(* IEC 61131-3 sources: ics_security/plc_ladder_logic/programs, 9 files *)

(* ---- led_ladder_logic_bomb.st ---- *)
PROGRAM part1c
  VAR
    Input0 AT %IX1.0 : BOOL;
    Output0 AT %QX1.0 : BOOL;
  END_VAR
  VAR
    TP0 : TP;
    Trigger0 : BOOL;
    Trigger1 : BOOL;
    CTU0 : CTU;
    TON0 : TON;
    SR0 : SR;
    R_TRIG1 : R_TRIG;
  END_VAR

  TP0(IN := Input0, PT := T#6s);
  Output0 := Input0 OR TP0.Q OR Trigger0 OR Trigger1;
  R_TRIG1(CLK := Input0);
  CTU0(CU := R_TRIG1.Q, PV := 6);
  Trigger0 := CTU0.Q;
  TON0(IN := Input0, PT := T#30s);
  SR0(S1 := TON0.Q);
  Trigger1 := SR0.Q1;
  Output0 := NOT(NOT(Input0) AND NOT(Trigger1) AND NOT(Trigger0));
END_PROGRAM

CONFIGURATION Config0

  RESOURCE Res0 ON PLC
    TASK task0(INTERVAL := T#20ms,PRIORITY := 0);
    PROGRAM instance0 WITH task0 : part1c;
  END_RESOURCE
END_CONFIGURATION

(* ---- led_loop.st ---- *)
PROGRAM part1b
  VAR
    Input0 AT %IX1.0 : BOOL;
    Output0 AT %QX1.0 : BOOL;
  END_VAR
  VAR
    TP0 : TP;
  END_VAR

  TP0(IN := Input0, PT := T#6s);
  Output0 := TP0.Q;
  Output0 := Input0;
  Output0 := NOT(NOT(Input0));
END_PROGRAM

CONFIGURATION Config0

  RESOURCE Res0 ON PLC
    TASK task0(INTERVAL := T#20ms,PRIORITY := 0);
    PROGRAM instance0 WITH task0 : part1b;
  END_RESOURCE
END_CONFIGURATION

(* ---- led_switch_activated.st ---- *)
PROGRAM part1a
  VAR
    Input0 AT %IX1.0 : BOOL;
    Input1 AT %IX1.1 : BOOL;
    Output0 AT %QX1.0 : BOOL;
    Output1 AT %QX1.1 : BOOL;
  END_VAR

  Output1 := Input0;
  Output0 := NOT(Input1);
END_PROGRAM

CONFIGURATION Config0

  RESOURCE Res0 ON PLC
    TASK task0(INTERVAL := T#20ms,PRIORITY := 0);
    PROGRAM instance0 WITH task0 : part1a;
  END_RESOURCE
END_CONFIGURATION

(* ---- robot_path.st ---- *)
PROGRAM part2
  VAR
    pos_x0 AT %IX0.0 : BOOL;
    pos_x1 AT %IX0.1 : BOOL;
    pos_x2 AT %IX0.2 : BOOL;
    pos_x3 AT %IX0.3 : BOOL;
  END_VAR
  VAR
    pos_x : UINT;
  END_VAR
  VAR
    pos_y0 AT %IX0.4 : BOOL;
    pos_y1 AT %IX0.5 : BOOL;
    pos_y2 AT %IX0.6 : BOOL;
    pos_y3 AT %IX0.7 : BOOL;
    target_x0 AT %IX1.0 : BOOL;
    target_x1 AT %IX1.1 : BOOL;
    target_x2 AT %IX1.2 : BOOL;
    target_x3 AT %IX1.3 : BOOL;
    target_y0 AT %IX1.4 : BOOL;
    target_y1 AT %IX1.5 : BOOL;
    target_y2 AT %IX1.6 : BOOL;
    target_y3 AT %IX1.7 : BOOL;
    dir_up AT %QX0.0 : BOOL;
    dir_down AT %QX0.1 : BOOL;
    dir_left AT %QX0.2 : BOOL;
    dir_right AT %QX0.3 : BOOL;
  END_VAR
  VAR
    BOOL_TO_UINT37_OUT : UINT;
    BOOL_TO_UINT3_OUT : UINT;
    MUL40_OUT : UINT;
    BOOL_TO_UINT4_OUT : UINT;
    MUL6_OUT : UINT;
    BOOL_TO_UINT5_OUT : UINT;
    MUL9_OUT : UINT;
    ADD42_OUT : UINT;
    BOOL_TO_UINT16_OUT : UINT;
    BOOL_TO_UINT27_OUT : UINT;
    MUL19_OUT : UINT;
    BOOL_TO_UINT15_OUT : UINT;
    MUL18_OUT : UINT;
    BOOL_TO_UINT32_OUT : UINT;
    MUL28_OUT : UINT;
    ADD31_OUT : UINT;
    GT43_OUT : BOOL;
    BOOL_TO_UINT76_OUT : UINT;
    BOOL_TO_UINT36_OUT : UINT;
    MUL77_OUT : UINT;
    BOOL_TO_UINT38_OUT : UINT;
    MUL48_OUT : UINT;
    BOOL_TO_UINT39_OUT : UINT;
    MUL51_OUT : UINT;
    ADD79_OUT : UINT;
    BOOL_TO_UINT58_OUT : UINT;
    BOOL_TO_UINT69_OUT : UINT;
    MUL61_OUT : UINT;
    BOOL_TO_UINT57_OUT : UINT;
    MUL60_OUT : UINT;
    BOOL_TO_UINT74_OUT : UINT;
    MUL70_OUT : UINT;
    ADD73_OUT : UINT;
    GT80_OUT : BOOL;
    LT44_OUT : BOOL;
    LT81_OUT : BOOL;
  END_VAR

  BOOL_TO_UINT37_OUT := BOOL_TO_UINT(pos_x0);
  BOOL_TO_UINT3_OUT := BOOL_TO_UINT(pos_x1);
  MUL40_OUT := MUL(BOOL_TO_UINT3_OUT, 2);
  BOOL_TO_UINT4_OUT := BOOL_TO_UINT(pos_x2);
  MUL6_OUT := MUL(BOOL_TO_UINT4_OUT, 2, 2);
  BOOL_TO_UINT5_OUT := BOOL_TO_UINT(pos_x3);
  MUL9_OUT := MUL(BOOL_TO_UINT5_OUT, 2, 2, 2);
  ADD42_OUT := ADD(BOOL_TO_UINT37_OUT, MUL40_OUT, MUL6_OUT, MUL9_OUT);
  BOOL_TO_UINT16_OUT := BOOL_TO_UINT(target_x0);
  BOOL_TO_UINT27_OUT := BOOL_TO_UINT(target_x1);
  MUL19_OUT := MUL(BOOL_TO_UINT27_OUT, 2);
  BOOL_TO_UINT15_OUT := BOOL_TO_UINT(target_x2);
  MUL18_OUT := MUL(BOOL_TO_UINT15_OUT, 2, 2);
  BOOL_TO_UINT32_OUT := BOOL_TO_UINT(target_x3);
  MUL28_OUT := MUL(BOOL_TO_UINT32_OUT, 2, 2, 2);
  ADD31_OUT := ADD(BOOL_TO_UINT16_OUT, MUL19_OUT, MUL18_OUT, MUL28_OUT);
  GT43_OUT := GT(ADD42_OUT, ADD31_OUT);
  dir_left := NOT(dir_right) AND NOT(dir_up) AND NOT(dir_down) AND GT43_OUT;
  BOOL_TO_UINT76_OUT := BOOL_TO_UINT(pos_y0);
  BOOL_TO_UINT36_OUT := BOOL_TO_UINT(pos_y1);
  MUL77_OUT := MUL(BOOL_TO_UINT36_OUT, 2);
  BOOL_TO_UINT38_OUT := BOOL_TO_UINT(pos_y2);
  MUL48_OUT := MUL(BOOL_TO_UINT38_OUT, 2, 2);
  BOOL_TO_UINT39_OUT := BOOL_TO_UINT(pos_y3);
  MUL51_OUT := MUL(BOOL_TO_UINT39_OUT, 2, 2, 2);
  ADD79_OUT := ADD(BOOL_TO_UINT76_OUT, MUL77_OUT, MUL48_OUT, MUL51_OUT);
  BOOL_TO_UINT58_OUT := BOOL_TO_UINT(target_y0);
  BOOL_TO_UINT69_OUT := BOOL_TO_UINT(target_y1);
  MUL61_OUT := MUL(BOOL_TO_UINT69_OUT, 2);
  BOOL_TO_UINT57_OUT := BOOL_TO_UINT(target_y2);
  MUL60_OUT := MUL(BOOL_TO_UINT57_OUT, 2, 2);
  BOOL_TO_UINT74_OUT := BOOL_TO_UINT(target_y3);
  MUL70_OUT := MUL(BOOL_TO_UINT74_OUT, 2, 2, 2);
  ADD73_OUT := ADD(BOOL_TO_UINT58_OUT, MUL61_OUT, MUL60_OUT, MUL70_OUT);
  GT80_OUT := GT(ADD79_OUT, ADD73_OUT);
  dir_down := NOT(dir_right) AND NOT(dir_left) AND NOT(dir_up) AND GT80_OUT;
  LT44_OUT := LT(ADD42_OUT, ADD31_OUT);
  dir_right := NOT(dir_left) AND NOT(dir_up) AND NOT(dir_down) AND LT44_OUT;
  LT81_OUT := LT(ADD79_OUT, ADD73_OUT);
  dir_up := NOT(dir_left) AND NOT(dir_right) AND NOT(dir_down) AND LT81_OUT;
END_PROGRAM

CONFIGURATION Config0

  RESOURCE Res0 ON PLC
    TASK task0(INTERVAL := T#20ms,PRIORITY := 0);
    PROGRAM instance0 WITH task0 : part2;
  END_RESOURCE
END_CONFIGURATION

(* ---- stirring_system.st ---- *)
PROGRAM part5a
  VAR
    MinLvlSensor AT %IX0.0 : BOOL;
    LowLvlSensor AT %IX0.1 : BOOL;
    MedLvlSensor AT %IX0.2 : BOOL;
    HighLvlSensor AT %IX0.3 : BOOL;
    InValve1_A AT %QX0.0 : BOOL;
    InValve2_B AT %QX0.1 : BOOL;
    InValve3_C AT %QX0.2 : BOOL;
    Blade AT %QX0.3 : BOOL;
    OutValve AT %QX0.4 : BOOL;
  END_VAR
  VAR
    State0 : BOOL := True;
    State1 : BOOL;
    State2 : BOOL;
    State3 : BOOL;
    State4 : BOOL;
    State5 : BOOL;
    State6 : BOOL;
    SR0 : SR;
    SR1 : SR;
    SR2 : SR;
    SR3 : SR;
    TON0 : TON;
    SR4 : SR;
    SR5 : SR;
    SR6 : SR;
    TON1 : TON;
  END_VAR

  InValve1_A := State1;
  SR0(S1 := State0, R := State2);
  State1 := SR0.Q1;
  InValve1_A := NOT(State0 OR State2 OR State3 OR State4 OR State5 OR State6);
  SR1(S1 := LowLvlSensor AND State1, R := State3);
  State2 := SR1.Q1;
  InValve2_B := State1 OR State2 OR State3;
  InValve2_B := NOT(State0 OR State4 OR State5 OR State6);
  SR2(S1 := MedLvlSensor AND State2, R := State4);
  State3 := SR2.Q1;
  InValve3_C := State3;
  InValve3_C := NOT(State0 OR State1 OR State2 OR State4 OR State5 OR State6);
  SR3(S1 := HighLvlSensor AND State3, R := State5);
  State4 := SR3.Q1;
  OutValve := State5 OR State6;
  OutValve := NOT(State0 OR State1 OR State2 OR State3 OR State4);
  TON0(IN := State4, PT := T#5s);
  SR4(S1 := TON0.Q, R := State6);
  State5 := SR4.Q1;
  Blade := State4 OR State5;
  Blade := NOT(State0 OR State1 OR State2 OR State3 OR State6);
  SR5(S1 := NOT(MinLvlSensor) AND State5, R := State0);
  State6 := SR5.Q1;
  TON1(IN := State6, PT := T#3s);
  SR6(S1 := TON1.Q, R := State1);
  State0 := SR6.Q1;
END_PROGRAM

CONFIGURATION Config0

  RESOURCE Res0 ON PLC
    TASK task0(INTERVAL := T#20ms,PRIORITY := 0);
    PROGRAM instance0 WITH task0 : part5a;
  END_RESOURCE
END_CONFIGURATION

(* ---- stirring_system_ladder_logic_bomb.st ---- *)
PROGRAM part5b
  VAR
    MinLvlSensor AT %IX0.0 : BOOL;
    LowLvlSensor AT %IX0.1 : BOOL;
    MedLvlSensor AT %IX0.2 : BOOL;
    HighLvlSensor AT %IX0.3 : BOOL;
    InValve1_A AT %QX0.0 : BOOL;
    InValve2_B AT %QX0.1 : BOOL;
    InValve3_C AT %QX0.2 : BOOL;
    Blade AT %QX0.3 : BOOL;
    OutValve AT %QX0.4 : BOOL;
  END_VAR
  VAR
    State0 : BOOL := True;
    State1 : BOOL;
    State2 : BOOL;
    State3 : BOOL;
    State4 : BOOL;
    State5 : BOOL;
    State6 : BOOL;
    SR0 : SR;
    SR1 : SR;
    SR2 : SR;
    SR3 : SR;
    TON0 : TON;
    SR4 : SR;
    SR5 : SR;
    SR6 : SR;
    TON1 : TON;
    Trigger : BOOL;
    CTU0 : CTU;
    SR7 : SR;
    R_TRIG1 : R_TRIG;
  END_VAR

  InValve1_A := State1;
  SR0(S1 := State0, R := State2);
  State1 := SR0.Q1;
  R_TRIG1(CLK := SR0.Q1);
  CTU0(CU := R_TRIG1.Q, PV := 4);
  SR7(S1 := CTU0.Q);
  Trigger := SR7.Q1;
  InValve1_A := NOT(State0 OR State2 OR State3 OR State4 OR State5 OR State6);
  SR1(S1 := LowLvlSensor AND State1, R := State3);
  State2 := SR1.Q1;
  InValve2_B := State1 OR State2 OR State3;
  InValve2_B := NOT(State0 OR State4 OR State5 OR State6);
  SR2(S1 := MedLvlSensor AND State2, R := State4);
  State3 := SR2.Q1;
  InValve3_C := State3;
  InValve3_C := NOT(State0 OR State1 OR State2 OR State4 OR State5 OR State6);
  SR3(S1 := HighLvlSensor AND State3, R := State5);
  State4 := SR3.Q1;
  OutValve := State5 OR State6;
  OutValve := NOT(State0 OR State1 OR State2 OR State3 OR State4);
  TON0(IN := State4, PT := T#5s);
  SR4(S1 := TON0.Q, R := State6);
  State5 := SR4.Q1;
  Blade := NOT(Trigger) AND State4 OR NOT(Trigger) AND State5 OR NOT(Trigger) AND State6 OR Trigger AND State1 OR Trigger AND State2 OR Trigger AND State3 OR Trigger AND State0;
  Blade := NOT(NOT(Trigger) AND State0 OR NOT(Trigger) AND State1 OR NOT(Trigger) AND State2 OR NOT(Trigger) AND State3 OR NOT(Trigger) AND State6 OR Trigger AND State4 OR Trigger AND State5);
  SR5(S1 := NOT(MinLvlSensor) AND State5, R := State0);
  State6 := SR5.Q1;
  TON1(IN := State6, PT := T#3s);
  SR6(S1 := TON1.Q, R := State1);
  State0 := SR6.Q1;
END_PROGRAM

CONFIGURATION Config0

  RESOURCE Res0 ON PLC
    TASK task0(INTERVAL := T#20ms,PRIORITY := 0);
    PROGRAM instance0 WITH task0 : part5b;
  END_RESOURCE
END_CONFIGURATION

(* ---- tank_balancer.st ---- *)
PROGRAM part4a
  VAR
    Tank1_LowLvlSensor AT %IX0.0 : BOOL;
    Tank1_MedLvlSensor AT %IX0.1 : BOOL;
    Tank1_HighLvlSensor AT %IX0.2 : BOOL;
    Tank2_LowLvlSensor AT %IX0.3 : BOOL;
    Tank2_MedLvlSensor AT %IX0.4 : BOOL;
    Tank2_HighLvlSensor AT %IX0.5 : BOOL;
    Tank3_LowLvlSensor AT %IX0.6 : BOOL;
    Tank3_MedLvlSensor AT %IX0.7 : BOOL;
    Tank3_HighLvlSensor AT %IX1.0 : BOOL;
    Tank4_LowLvlSensor AT %IX1.1 : BOOL;
    Tank4_MedLvlSensor AT %IX1.2 : BOOL;
    Tank4_HighLvlSensor AT %IX1.3 : BOOL;
    Tank1_OutValve AT %QX0.0 : BOOL;
    Tank2_OutValve AT %QX0.1 : BOOL;
    Tank3_OutValve AT %QX0.2 : BOOL;
    Tank4_OutValve AT %QX0.3 : BOOL;
  END_VAR

  Tank1_OutValve := NOT(NOT(Tank1_MedLvlSensor) AND Tank1_LowLvlSensor OR NOT(Tank1_LowLvlSensor));
  Tank1_OutValve := Tank1_MedLvlSensor;
  Tank2_OutValve := NOT(NOT(Tank2_MedLvlSensor) AND Tank2_LowLvlSensor OR NOT(Tank2_LowLvlSensor));
  Tank2_OutValve := Tank2_MedLvlSensor;
  Tank3_OutValve := NOT(NOT(Tank3_MedLvlSensor) AND Tank3_LowLvlSensor OR NOT(Tank3_LowLvlSensor));
  Tank3_OutValve := Tank3_MedLvlSensor;
  Tank4_OutValve := NOT(NOT(Tank4_MedLvlSensor) AND Tank4_LowLvlSensor OR NOT(Tank4_LowLvlSensor));
  Tank4_OutValve := Tank4_MedLvlSensor;
END_PROGRAM

CONFIGURATION Config0

  RESOURCE Res0 ON PLC
    TASK task0(INTERVAL := T#20ms,PRIORITY := 0);
    PROGRAM instance0 WITH task0 : part4a;
  END_RESOURCE
END_CONFIGURATION

(* ---- tank_balancer_ladder_logic_bomb.st ---- *)
PROGRAM part4b
  VAR
    Tank1_LowLvlSensor AT %IX0.0 : BOOL;
    Tank1_MedLvlSensor AT %IX0.1 : BOOL;
    Tank1_HighLvlSensor AT %IX0.2 : BOOL;
    Tank2_LowLvlSensor AT %IX0.3 : BOOL;
    Tank2_MedLvlSensor AT %IX0.4 : BOOL;
    Tank2_HighLvlSensor AT %IX0.5 : BOOL;
    Tank3_LowLvlSensor AT %IX0.6 : BOOL;
    Tank3_MedLvlSensor AT %IX0.7 : BOOL;
    Tank3_HighLvlSensor AT %IX1.0 : BOOL;
    Tank4_LowLvlSensor AT %IX1.1 : BOOL;
    Tank4_MedLvlSensor AT %IX1.2 : BOOL;
    Tank4_HighLvlSensor AT %IX1.3 : BOOL;
    Tank1_OutValve AT %QX0.0 : BOOL;
    Tank2_OutValve AT %QX0.1 : BOOL;
    Tank3_OutValve AT %QX0.2 : BOOL;
    Tank4_OutValve AT %QX0.3 : BOOL;
  END_VAR
  VAR
    Trigger : BOOL;
    TON0 : TON;
  END_VAR

  Tank1_OutValve := NOT(NOT(Tank1_MedLvlSensor) AND Tank1_LowLvlSensor OR NOT(Tank1_LowLvlSensor));
  TON0(IN := Tank2_LowLvlSensor, PT := T#30s);
  Trigger := TON0.Q;
  Tank1_OutValve := Tank1_MedLvlSensor;
  Tank2_OutValve := NOT(NOT(Tank2_MedLvlSensor) AND Tank2_LowLvlSensor OR NOT(Tank2_LowLvlSensor) OR Trigger);
  Tank2_OutValve := NOT(Trigger) AND Tank2_MedLvlSensor;
  Tank3_OutValve := NOT(NOT(Tank3_MedLvlSensor) AND Tank3_LowLvlSensor OR NOT(Tank3_LowLvlSensor));
  Tank3_OutValve := Tank3_MedLvlSensor;
  Tank4_OutValve := NOT(NOT(Tank4_MedLvlSensor) AND Tank4_LowLvlSensor OR NOT(Tank4_LowLvlSensor));
  Tank4_OutValve := Tank4_MedLvlSensor;
END_PROGRAM

CONFIGURATION Config0

  RESOURCE Res0 ON PLC
    TASK task0(INTERVAL := T#20ms,PRIORITY := 0);
    PROGRAM instance0 WITH task0 : part4b;
  END_RESOURCE
END_CONFIGURATION

(* ---- traffic_light.st ---- *)
PROGRAM part3
  VAR
    VehSensor AT %IX0.0 : BOOL;
    PedXINGButton AT %IX0.1 : BOOL;
    VehRedLight AT %QX0.0 : BOOL;
    VehYellowLight AT %QX0.1 : BOOL;
    VehGreenLight AT %QX0.2 : BOOL;
    PedRedLight AT %QX0.3 : BOOL;
    PedGreenLight AT %QX0.4 : BOOL;
  END_VAR
  VAR
    State0 : BOOL := True;
    State1 : BOOL;
    State2 : BOOL;
    State3 : BOOL;
    TP0 : TP;
    SR0 : SR;
    SR1 : SR;
    TON0 : TON;
    TON1 : TON;
    SR2 : SR;
    SR3 : SR;
    TON2 : TON;
  END_VAR

  VehGreenLight := State0;
  TP0(IN := PedXINGButton AND State0, PT := T#1s);
  SR0(S1 := NOT(VehSensor) AND TP0.Q, R := State2);
  State1 := SR0.Q1;
  VehGreenLight := NOT(State1 OR State2 OR State3);
  VehYellowLight := State1;
  VehYellowLight := NOT(State0 OR State2 OR State3);
  TON1(IN := State1, PT := T#3s);
  SR2(S1 := TON1.Q, R := State3);
  State2 := SR2.Q1;
  VehRedLight := State1 OR State2 OR State3;
  VehRedLight := NOT(State0 OR State1);
  PedGreenLight := State2;
  TON2(IN := State2, PT := T#15s);
  SR3(S1 := TON2.Q, R := State0);
  State3 := SR3.Q1;
  PedGreenLight := NOT(State0 OR State1 OR State3);
  PedRedLight := State0 OR State1 OR State3;
  PedRedLight := NOT(State2);
  TON0(IN := State3, PT := T#1s);
  SR1(S1 := State1, R := TON0.Q);
  State0 := NOT(SR1.Q1);
END_PROGRAM

CONFIGURATION Config0

  RESOURCE Res0 ON PLC
    TASK task0(INTERVAL := T#20ms,PRIORITY := 0);
    PROGRAM instance0 WITH task0 : part3;
  END_RESOURCE
END_CONFIGURATION
